Fanuc KAREL source: kt00157.KL

-- PROVISIONAL review KL for V770-1; original PC SHA256 5900e96a64e9c8d72d96b980e561b96e61bb12f30f8bfbd177e4fe2525148cec
-- Incomplete behavior may be omitted. Consult companion uncertainty JSON. Do not deploy.
PROGRAM KT00157
%NOLOCKGROUP
VAR
  OUT : INTEGER
-- UNRESOLVED_DECL H1 type=002017
-- UNRESOLVED_DECL Y2 type=002018
BEGIN
  -- UNRESOLVED_PC offsets 5-19; opcodes 2E,22,9D,33,B4
  -- UNRESOLVED_PC offsets 24-38; opcodes 2E,22,9D,33,B2
  -- UNRESOLVED_PC offsets 43-68; opcodes 22,9D,33,B3,22,9D,33,B1,55,23
  -- UNRESOLVED_PC offsets 73-77; opcodes 7F
END KT00157
